Staubli VAL3: onStop.pgx

public program onStop(string& x_sItem[])
begin
end
